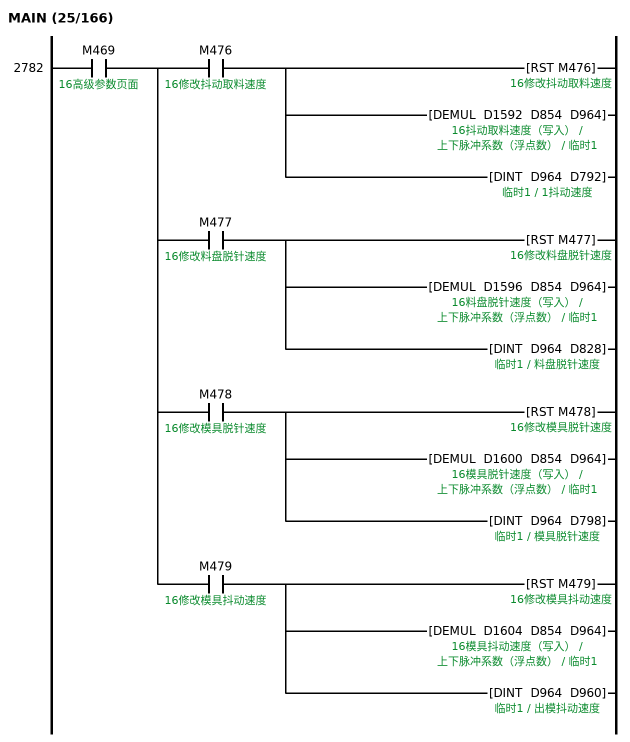
[picture p24: ladder of MAIN, rungs at steps 2782 to 2782]
2782  LD      M469  ; 16高级参数页面
      MPS
      AND     M476  ; 16修改抖动取料速度
      RST     M476  ; 16修改抖动取料速度
      DEMUL   D1592 D854 D964  ; 16抖动取料速度（写入）
      DINT    D964 D792
      MRD
      AND     M477  ; 16修改料盘脱针速度
      RST     M477  ; 16修改料盘脱针速度
      DEMUL   D1596 D854 D964  ; 16料盘脱针速度（写入）
      DINT    D964 D828
      MRD
      AND     M478  ; 16修改模具脱针速度
      RST     M478  ; 16修改模具脱针速度
      DEMUL   D1600 D854 D964  ; 16模具脱针速度（写入）
      DINT    D964 D798
      MPP
      AND     M479  ; 16修改模具抖动速度
      RST     M479  ; 16修改模具抖动速度
      DEMUL   D1604 D854 D964  ; 16模具抖动速度（写入）
      DINT    D964 D960
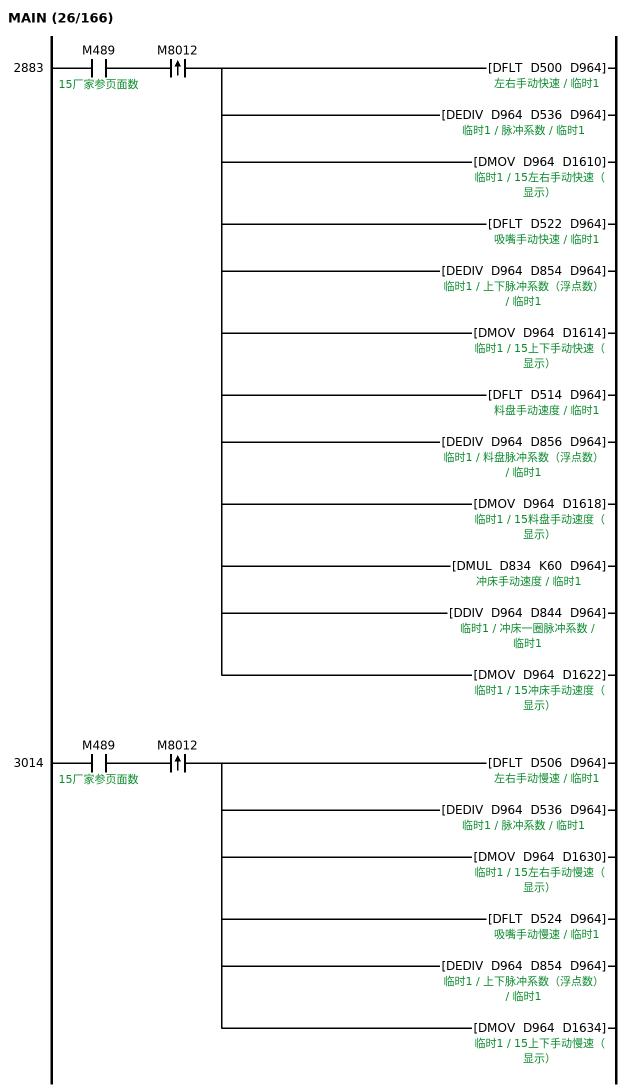
2883  LD      M489  ; 15厂家参页面数
      ANDP    M8012
      DFLT    D500 D964  ; 左右手动快速
      DEDIV   D964 D536 D964
      DMOV    D964 D1610  ; 15左右手动快速（显示）
      DFLT    D522 D964  ; 吸嘴手动快速
      DEDIV   D964 D854 D964
      DMOV    D964 D1614  ; 15上下手动快速（显示）
      DFLT    D514 D964  ; 料盘手动速度
      DEDIV   D964 D856 D964
      DMOV    D964 D1618  ; 15料盘手动速度（显示）
      DMUL    D834 K60 D964  ; 冲床手动速度
      DDIV    D964 D844 D964
      DMOV    D964 D1622  ; 15冲床手动速度（显示）
3014  LD      M489  ; 15厂家参页面数
      ANDP    M8012
      DFLT    D506 D964  ; 左右手动慢速
      DEDIV   D964 D536 D964
      DMOV    D964 D1630  ; 15左右手动慢速（显示）
      DFLT    D524 D964  ; 吸嘴手动慢速
      DEDIV   D964 D854 D964
      DMOV    D964 D1634  ; 15上下手动慢速（显示）
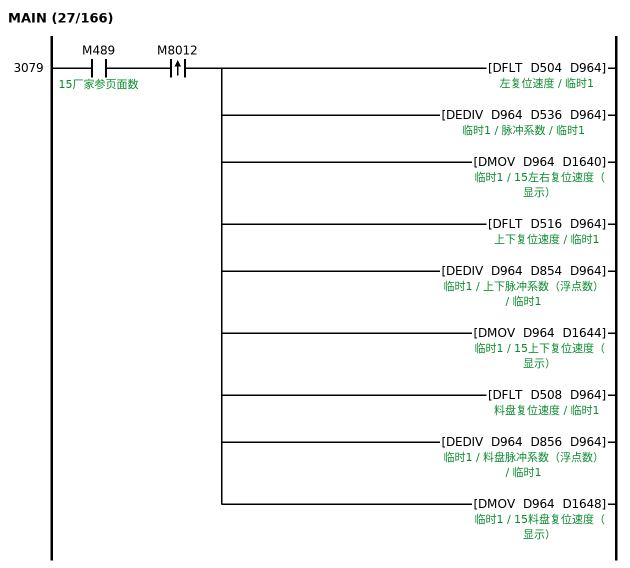
3079  LD      M489  ; 15厂家参页面数
      ANDP    M8012
      DFLT    D504 D964  ; 左复位速度
      DEDIV   D964 D536 D964
      DMOV    D964 D1640  ; 15左右复位速度（显示）
      DFLT    D516 D964  ; 上下复位速度
      DEDIV   D964 D854 D964
      DMOV    D964 D1644  ; 15上下复位速度（显示）
      DFLT    D508 D964  ; 料盘复位速度
      DEDIV   D964 D856 D964
      DMOV    D964 D1648  ; 15料盘复位速度（显示）
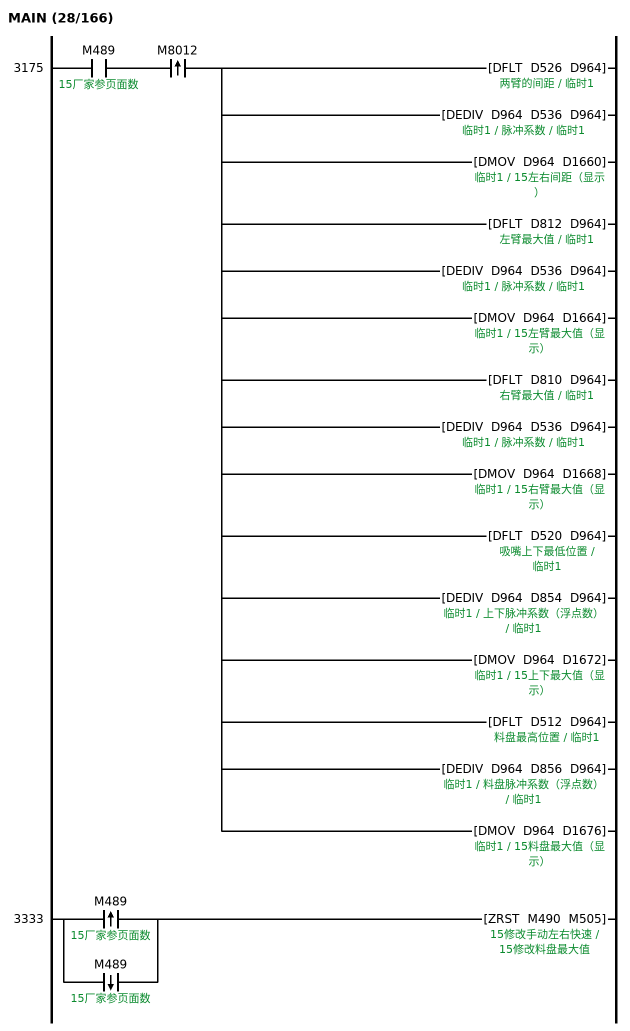
3175  LD      M489  ; 15厂家参页面数
      ANDP    M8012
      DFLT    D526 D964
      DEDIV   D964 D536 D964
      DMOV    D964 D1660  ; 15左右间距（显示）
      DFLT    D812 D964  ; 左臂最大值
      DEDIV   D964 D536 D964
      DMOV    D964 D1664  ; 15左臂最大值（显示）
      DFLT    D810 D964  ; 右臂最大值
      DEDIV   D964 D536 D964
      DMOV    D964 D1668  ; 15右臂最大值（显示）
      DFLT    D520 D964  ; 吸嘴上下最低位置
      DEDIV   D964 D854 D964
      DMOV    D964 D1672  ; 15上下最大值（显示）
      DFLT    D512 D964  ; 料盘最高位置
      DEDIV   D964 D856 D964
      DMOV    D964 D1676  ; 15料盘最大值（显示）
3333  LDP     M489  ; 15厂家参页面数
      ORF     M489  ; 15厂家参页面数
      ZRST    M490 M505  ; 15修改手动左右快速 / 15修改料盘最大值
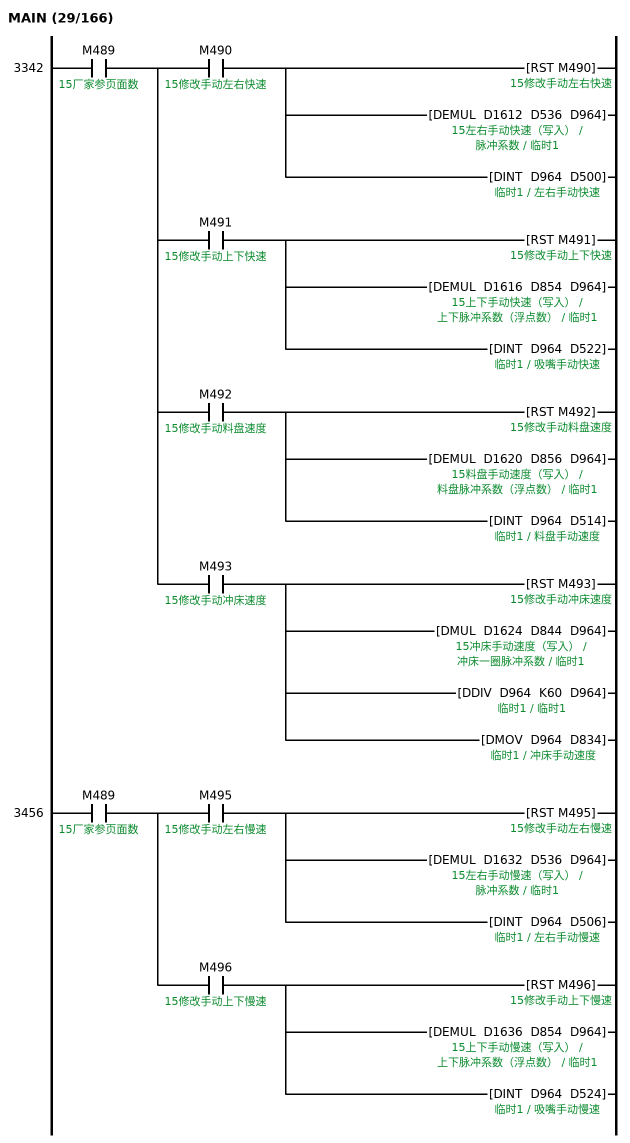
3342  LD      M489  ; 15厂家参页面数
      MPS
      AND     M490  ; 15修改手动左右快速
      RST     M490  ; 15修改手动左右快速
      DEMUL   D1612 D536 D964  ; 15左右手动快速（写入）
      DINT    D964 D500
      MRD
      AND     M491  ; 15修改手动上下快速
      RST     M491  ; 15修改手动上下快速
      DEMUL   D1616 D854 D964  ; 15上下手动快速（写入）
      DINT    D964 D522
      MRD
      AND     M492  ; 15修改手动料盘速度
      RST     M492  ; 15修改手动料盘速度
      DEMUL   D1620 D856 D964  ; 15料盘手动速度（写入）
      DINT    D964 D514
      MPP
      AND     M493  ; 15修改手动冲床速度
      RST     M493  ; 15修改手动冲床速度
      DMUL    D1624 D844 D964  ; 15冲床手动速度（写入）
      DDIV    D964 K60 D964
      DMOV    D964 D834
3456  LD      M489  ; 15厂家参页面数
      MPS
      AND     M495  ; 15修改手动左右慢速
      RST     M495  ; 15修改手动左右慢速
      DEMUL   D1632 D536 D964  ; 15左右手动慢速（写入）
      DINT    D964 D506
      MPP
      AND     M496  ; 15修改手动上下慢速
      RST     M496  ; 15修改手动上下慢速
      DEMUL   D1636 D854 D964  ; 15上下手动慢速（写入）
      DINT    D964 D524
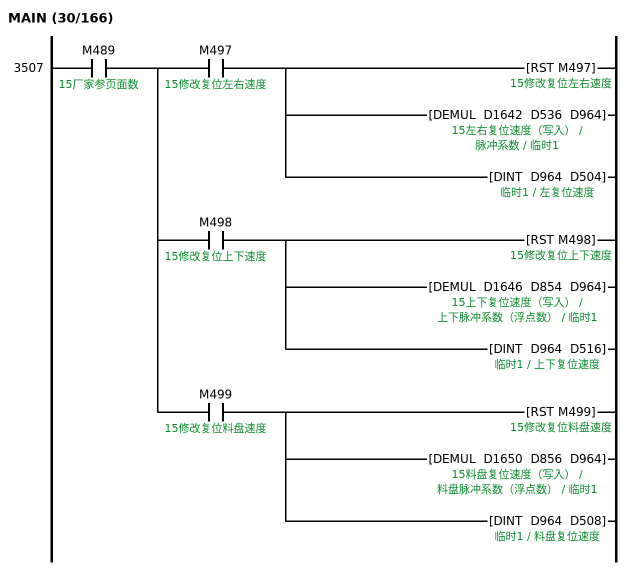
3507  LD      M489  ; 15厂家参页面数
      MPS
      AND     M497  ; 15修改复位左右速度
      RST     M497  ; 15修改复位左右速度
      DEMUL   D1642 D536 D964  ; 15左右复位速度（写入）
      DINT    D964 D504
      MRD
      AND     M498  ; 15修改复位上下速度
      RST     M498  ; 15修改复位上下速度
      DEMUL   D1646 D854 D964  ; 15上下复位速度（写入）
      DINT    D964 D516
      MPP
      AND     M499  ; 15修改复位料盘速度
      RST     M499  ; 15修改复位料盘速度
      DEMUL   D1650 D856 D964  ; 15料盘复位速度（写入）
      DINT    D964 D508
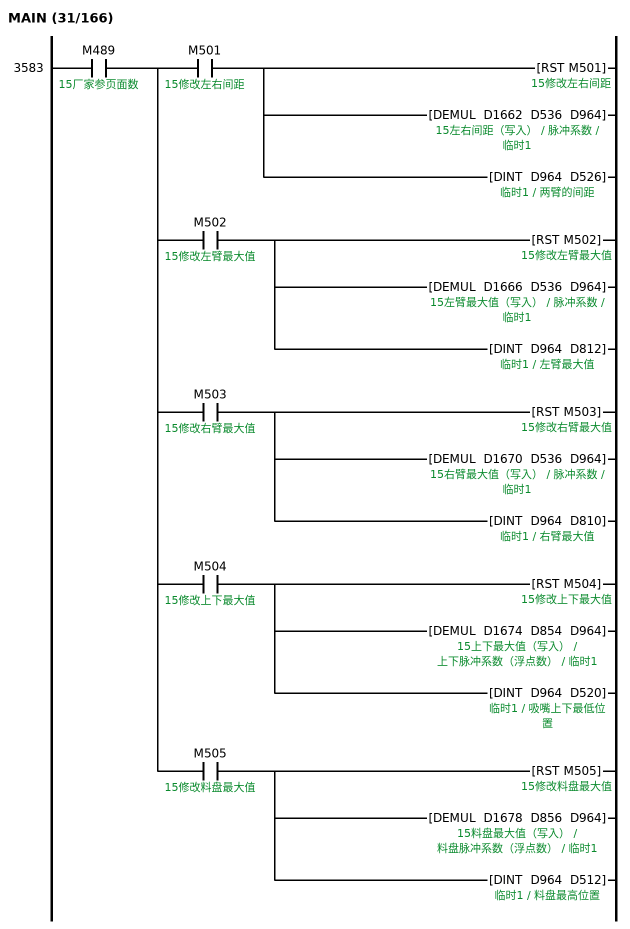
3583  LD      M489  ; 15厂家参页面数
      MPS
      AND     M501  ; 15修改左右间距
      RST     M501  ; 15修改左右间距
      DEMUL   D1662 D536 D964  ; 15左右间距（写入）
      DINT    D964 D526
      MRD
      AND     M502  ; 15修改左臂最大值
      RST     M502  ; 15修改左臂最大值
      DEMUL   D1666 D536 D964  ; 15左臂最大值（写入）
      DINT    D964 D812
      MRD
      AND     M503  ; 15修改右臂最大值
      RST     M503  ; 15修改右臂最大值
      DEMUL   D1670 D536 D964  ; 15右臂最大值（写入）
      DINT    D964 D810
      MRD
      AND     M504  ; 15修改上下最大值
      RST     M504  ; 15修改上下最大值
      DEMUL   D1674 D854 D964  ; 15上下最大值（写入）
      DINT    D964 D520
      MPP
      AND     M505  ; 15修改料盘最大值
      RST     M505  ; 15修改料盘最大值
      DEMUL   D1678 D856 D964  ; 15料盘最大值（写入）
      DINT    D964 D512
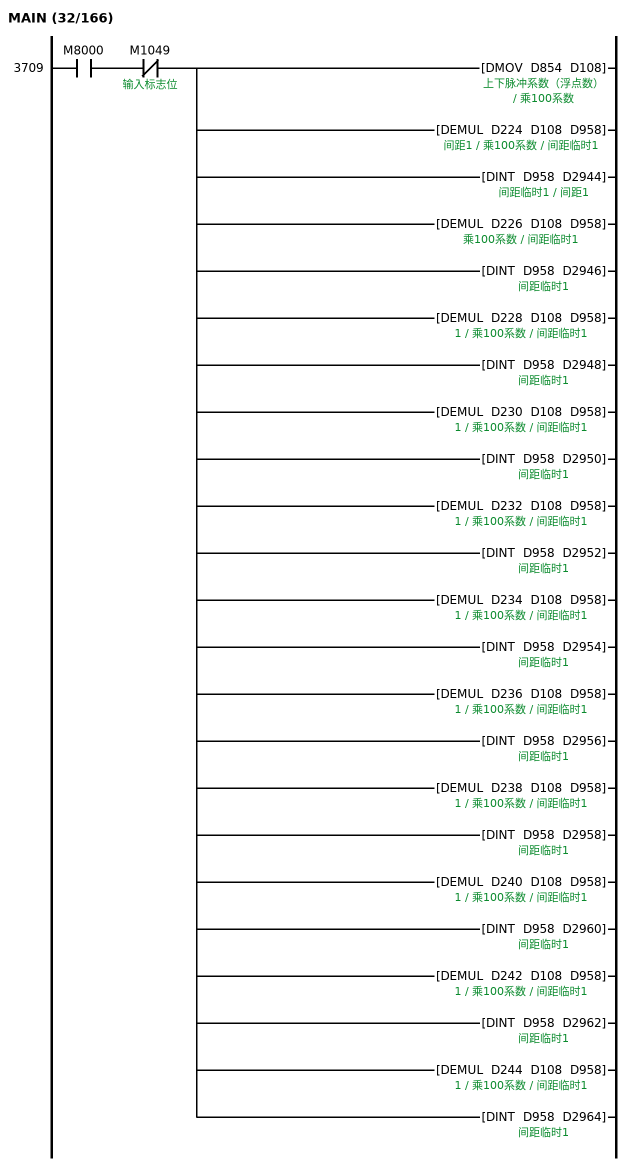
3709  LD      M8000
      ANI     M1049  ; 输入标志位
      DMOV    D854 D108  ; 乘100系数
      DEMUL   D224 D108 D958  ; 间距1 / 间距临时1
      DINT    D958 D2944  ; 间距1
      DEMUL   D226 D108 D958
      DINT    D958 D2946
      DEMUL   D228 D108 D958  ; 1
      DINT    D958 D2948
      DEMUL   D230 D108 D958  ; 1
      DINT    D958 D2950
      DEMUL   D232 D108 D958  ; 1
      DINT    D958 D2952
      DEMUL   D234 D108 D958  ; 1
      DINT    D958 D2954
      DEMUL   D236 D108 D958  ; 1
      DINT    D958 D2956
      DEMUL   D238 D108 D958  ; 1
      DINT    D958 D2958
      DEMUL   D240 D108 D958  ; 1
      DINT    D958 D2960
      DEMUL   D242 D108 D958  ; 1
      DINT    D958 D2962
      DEMUL   D244 D108 D958  ; 1
      DINT    D958 D2964
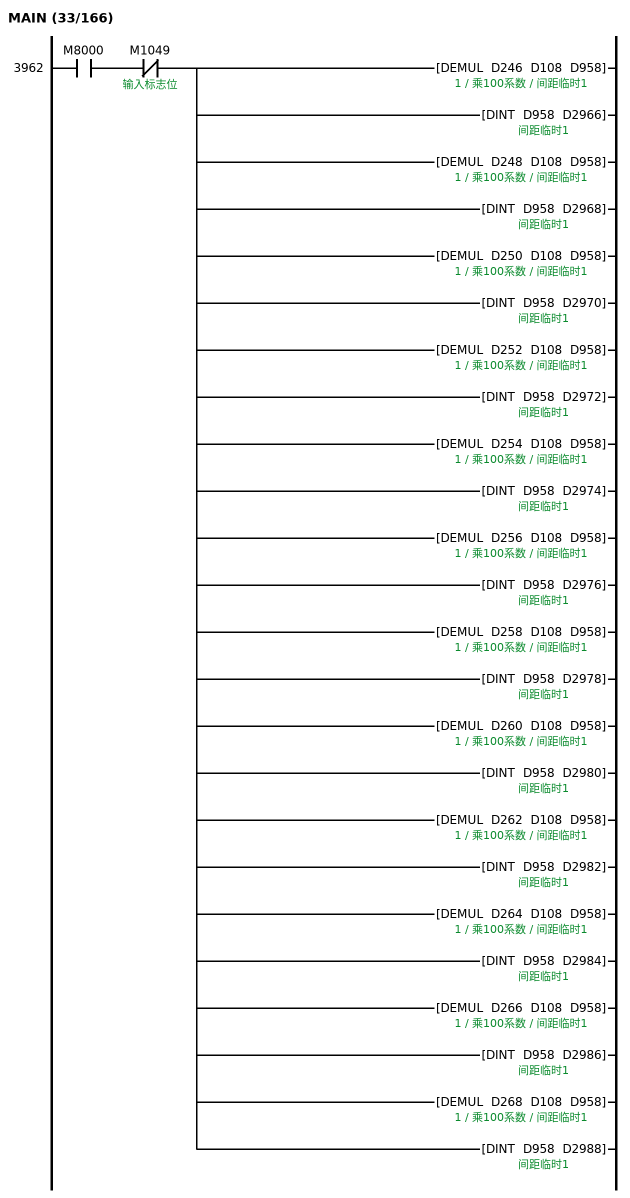
3962  LD      M8000
      ANI     M1049  ; 输入标志位
      DEMUL   D246 D108 D958  ; 1
      DINT    D958 D2966
      DEMUL   D248 D108 D958  ; 1
      DINT    D958 D2968
      DEMUL   D250 D108 D958  ; 1
      DINT    D958 D2970
      DEMUL   D252 D108 D958  ; 1
      DINT    D958 D2972
      DEMUL   D254 D108 D958  ; 1
      DINT    D958 D2974
      DEMUL   D256 D108 D958  ; 1
      DINT    D958 D2976
      DEMUL   D258 D108 D958  ; 1
      DINT    D958 D2978
      DEMUL   D260 D108 D958  ; 1
      DINT    D958 D2980
      DEMUL   D262 D108 D958  ; 1
      DINT    D958 D2982
      DEMUL   D264 D108 D958  ; 1
      DINT    D958 D2984
      DEMUL   D266 D108 D958  ; 1
      DINT    D958 D2986
      DEMUL   D268 D108 D958  ; 1
      DINT    D958 D2988
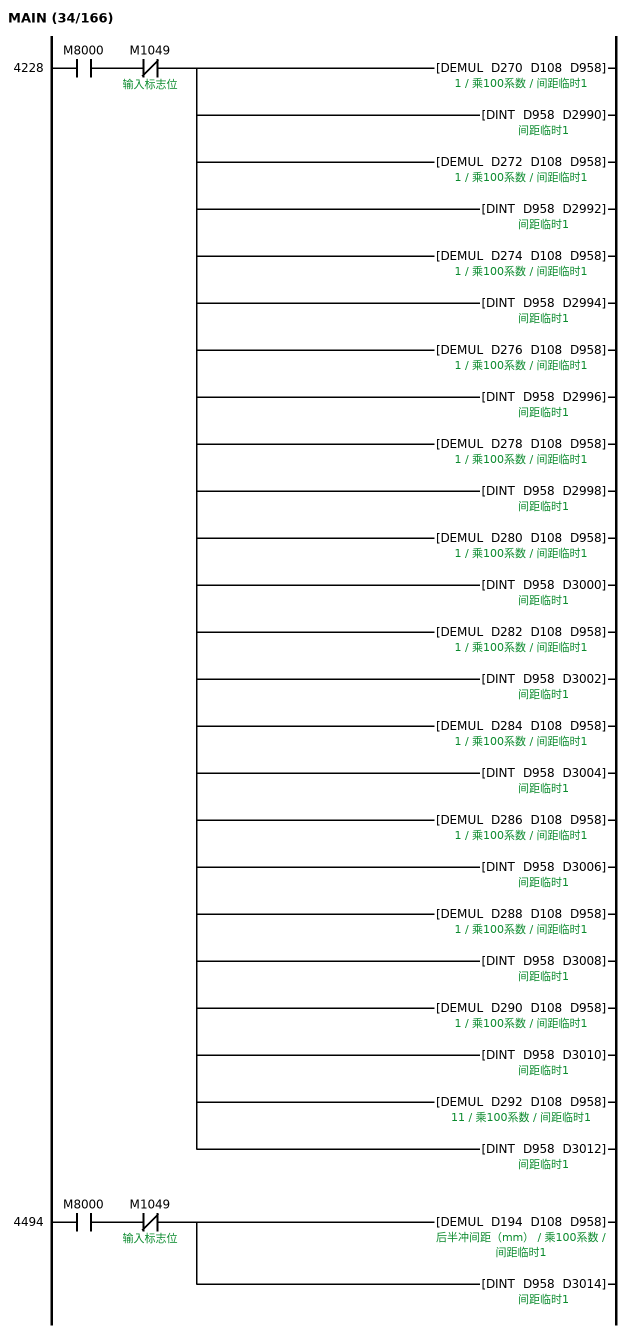
4228  LD      M8000
      ANI     M1049  ; 输入标志位
      DEMUL   D270 D108 D958  ; 1
      DINT    D958 D2990
      DEMUL   D272 D108 D958  ; 1
      DINT    D958 D2992
      DEMUL   D274 D108 D958  ; 1
      DINT    D958 D2994
      DEMUL   D276 D108 D958  ; 1
      DINT    D958 D2996
      DEMUL   D278 D108 D958  ; 1
      DINT    D958 D2998
      DEMUL   D280 D108 D958  ; 1
      DINT    D958 D3000
      DEMUL   D282 D108 D958  ; 1
      DINT    D958 D3002
      DEMUL   D284 D108 D958  ; 1
      DINT    D958 D3004
      DEMUL   D286 D108 D958  ; 1
      DINT    D958 D3006
      DEMUL   D288 D108 D958  ; 1
      DINT    D958 D3008
      DEMUL   D290 D108 D958  ; 1
      DINT    D958 D3010
      DEMUL   D292 D108 D958  ; 11
      DINT    D958 D3012
4494  LD      M8000
      ANI     M1049  ; 输入标志位
      DEMUL   D194 D108 D958
      DINT    D958 D3014
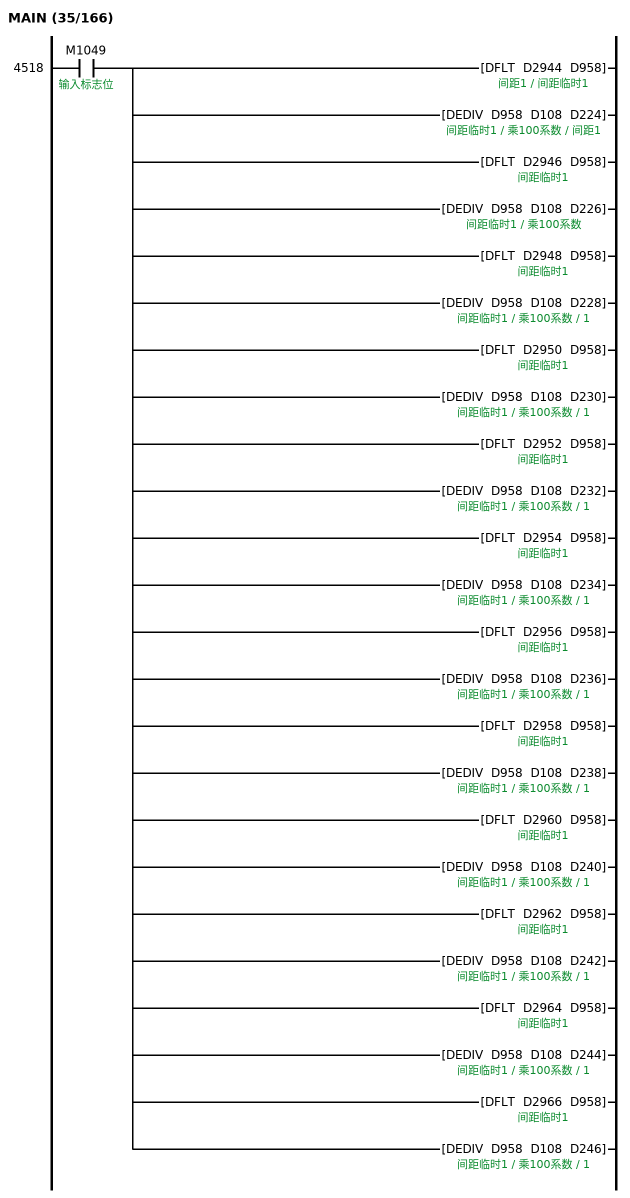
4518  LD      M1049  ; 输入标志位
      DFLT    D2944 D958
      DEDIV   D958 D108 D224
      DFLT    D2946 D958
      DEDIV   D958 D108 D226
      DFLT    D2948 D958
      DEDIV   D958 D108 D228
      DFLT    D2950 D958
      DEDIV   D958 D108 D230
      DFLT    D2952 D958
      DEDIV   D958 D108 D232
      DFLT    D2954 D958
      DEDIV   D958 D108 D234
      DFLT    D2956 D958
      DEDIV   D958 D108 D236
      DFLT    D2958 D958
      DEDIV   D958 D108 D238
      DFLT    D2960 D958
      DEDIV   D958 D108 D240
      DFLT    D2962 D958
      DEDIV   D958 D108 D242
      DFLT    D2964 D958
      DEDIV   D958 D108 D244
      DFLT    D2966 D958
      DEDIV   D958 D108 D246
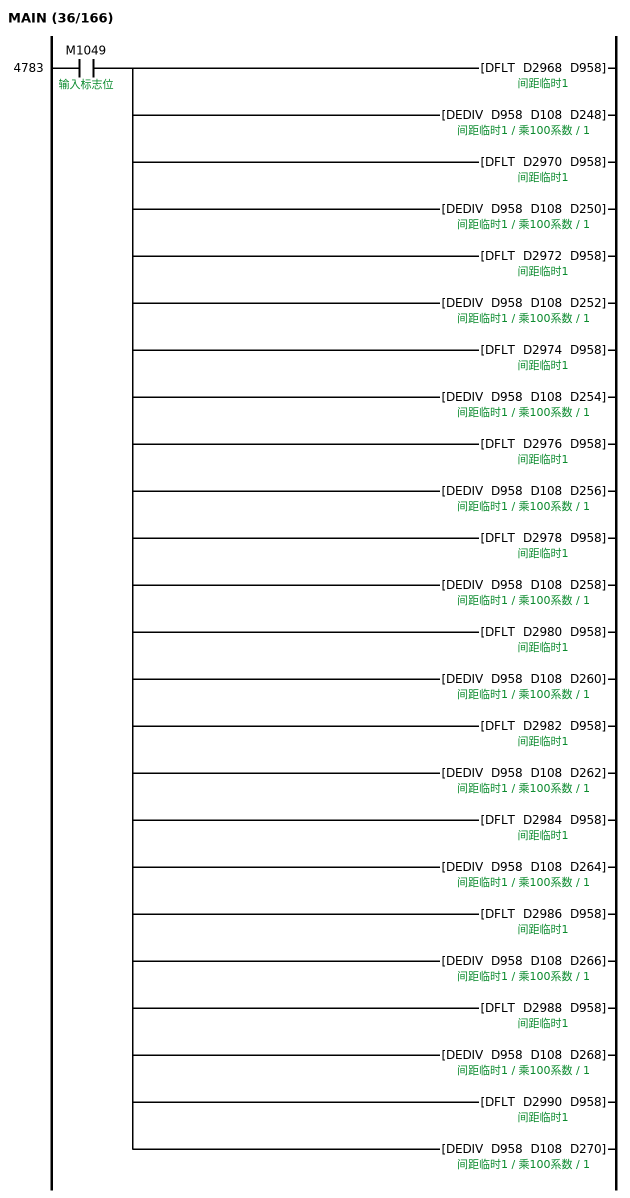
4783  LD      M1049  ; 输入标志位
      DFLT    D2968 D958
      DEDIV   D958 D108 D248
      DFLT    D2970 D958
      DEDIV   D958 D108 D250
      DFLT    D2972 D958
      DEDIV   D958 D108 D252
      DFLT    D2974 D958
      DEDIV   D958 D108 D254
      DFLT    D2976 D958
      DEDIV   D958 D108 D256
      DFLT    D2978 D958
      DEDIV   D958 D108 D258
      DFLT    D2980 D958
      DEDIV   D958 D108 D260
      DFLT    D2982 D958
      DEDIV   D958 D108 D262
      DFLT    D2984 D958
      DEDIV   D958 D108 D264
      DFLT    D2986 D958
      DEDIV   D958 D108 D266
      DFLT    D2988 D958
      DEDIV   D958 D108 D268
      DFLT    D2990 D958
      DEDIV   D958 D108 D270
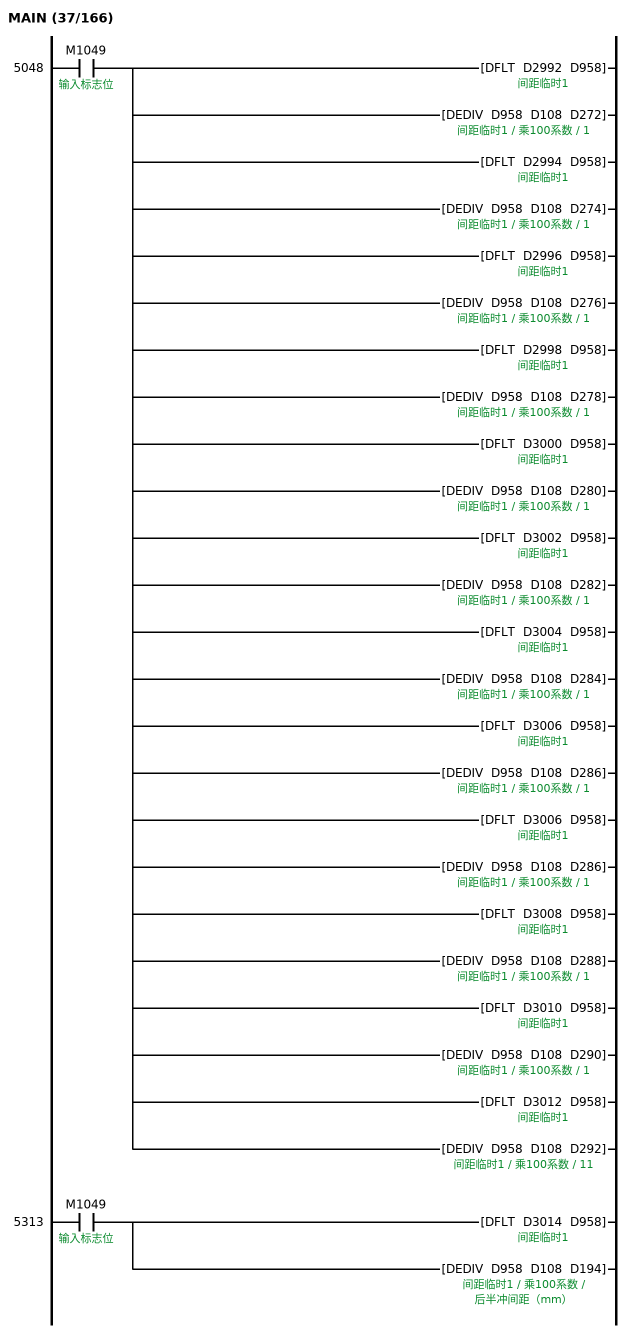
5048  LD      M1049  ; 输入标志位
      DFLT    D2992 D958
      DEDIV   D958 D108 D272
      DFLT    D2994 D958
      DEDIV   D958 D108 D274
      DFLT    D2996 D958
      DEDIV   D958 D108 D276
      DFLT    D2998 D958
      DEDIV   D958 D108 D278
      DFLT    D3000 D958
      DEDIV   D958 D108 D280
      DFLT    D3002 D958
      DEDIV   D958 D108 D282
      DFLT    D3004 D958
      DEDIV   D958 D108 D284
      DFLT    D3006 D958
      DEDIV   D958 D108 D286
      DFLT    D3006 D958
      DEDIV   D958 D108 D286
      DFLT    D3008 D958
      DEDIV   D958 D108 D288
      DFLT    D3010 D958
      DEDIV   D958 D108 D290
      DFLT    D3012 D958
      DEDIV   D958 D108 D292
5313  LD      M1049  ; 输入标志位
      DFLT    D3014 D958
      DEDIV   D958 D108 D194
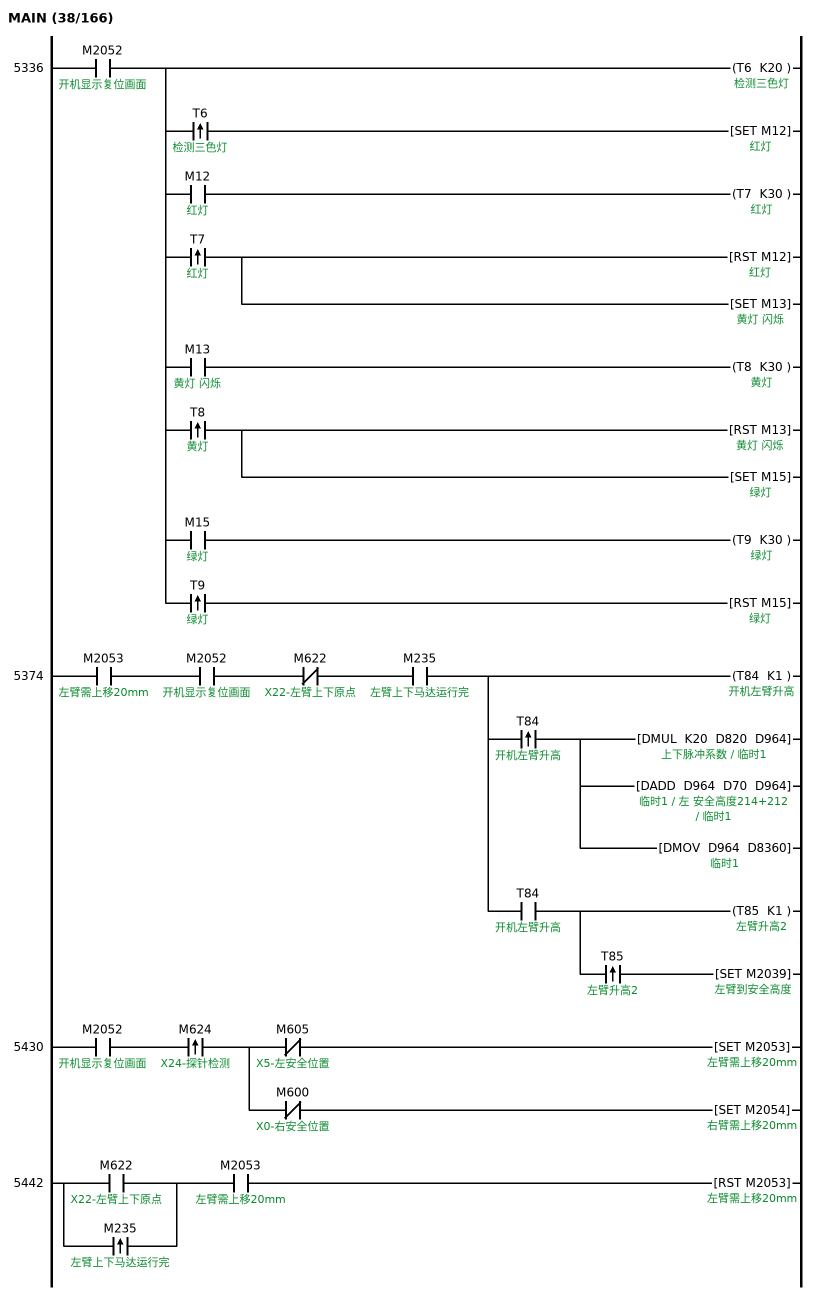
5336  LD      M2052  ; 开机显示复位画面
      OUT     T6 K20  ; 检测三色灯
      MPS
      ANDP    T6  ; 检测三色灯
      SET     M12  ; 红灯
      MRD
      AND     M12  ; 红灯
      OUT     T7 K30  ; 红灯
      MRD
      ANDP    T7  ; 红灯
      RST     M12  ; 红灯
      SET     M13  ; 黄灯 闪烁
      MRD
      AND     M13  ; 黄灯 闪烁
      OUT     T8 K30  ; 黄灯
      MRD
      ANDP    T8  ; 黄灯
      RST     M13  ; 黄灯 闪烁
      SET     M15  ; 绿灯
      MRD
      AND     M15  ; 绿灯
      OUT     T9 K30  ; 绿灯
      MPP
      ANDP    T9  ; 绿灯
      RST     M15  ; 绿灯
5374  LD      M2053  ; 左臂需上移20mm
      AND     M2052  ; 开机显示复位画面
      ANI     M622  ; X22-左臂上下原点
      AND     M235  ; 左臂上下马达运行完
      OUT     T84 K1  ; 开机左臂升高
      MPS
      ANDP    T84  ; 开机左臂升高
      DMUL    K20 D820 D964
      DADD    D964 D70 D964
      DMOV    D964 D8360
      MPP
      AND     T84  ; 开机左臂升高
      OUT     T85 K1  ; 左臂升高2
      ANDP    T85  ; 左臂升高2
      SET     M2039  ; 左臂到安全高度
5430  LD      M2052  ; 开机显示复位画面
      ANDP    M624  ; X24-探针检测
      MPS
      ANI     M605  ; X5-左安全位置
      SET     M2053  ; 左臂需上移20mm
      MPP
      ANI     M600  ; X0-右安全位置
      SET     M2054  ; 右臂需上移20mm
5442  LD      M622  ; X22-左臂上下原点
      ORP     M235  ; 左臂上下马达运行完
      AND     M2053  ; 左臂需上移20mm
      RST     M2053  ; 左臂需上移20mm
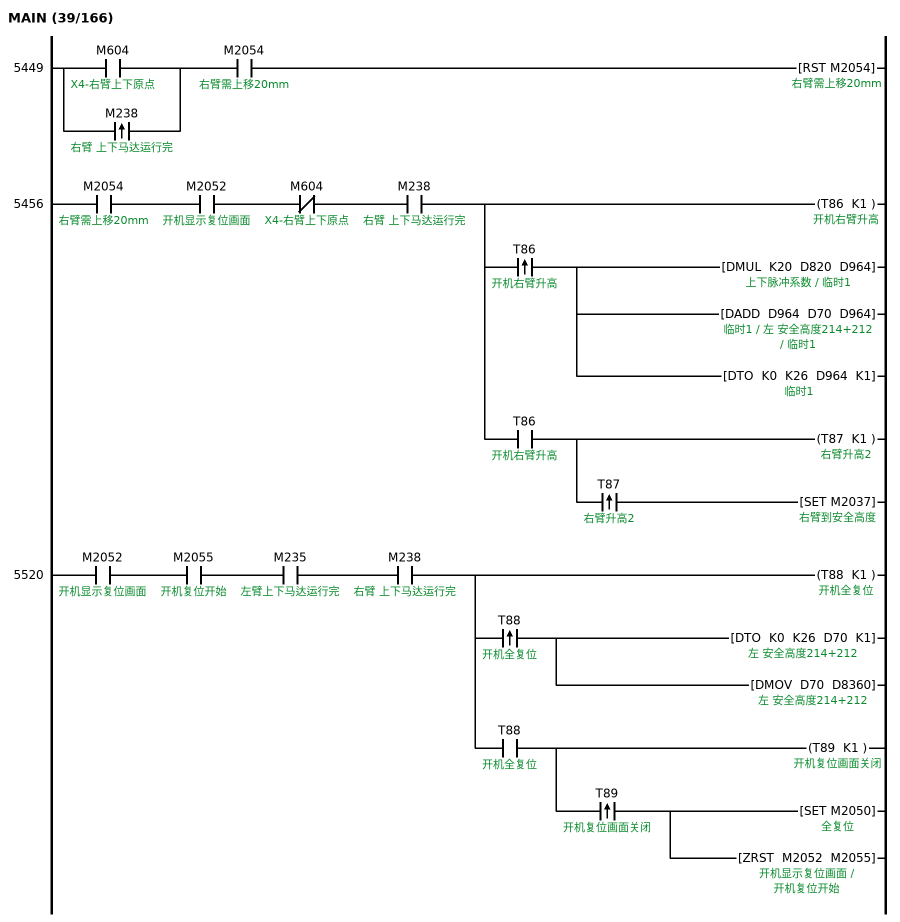
5449  LD      M604  ; X4-右臂上下原点
      ORP     M238  ; 右臂 上下马达运行完
      AND     M2054  ; 右臂需上移20mm
      RST     M2054  ; 右臂需上移20mm
5456  LD      M2054  ; 右臂需上移20mm
      AND     M2052  ; 开机显示复位画面
      ANI     M604  ; X4-右臂上下原点
      AND     M238  ; 右臂 上下马达运行完
      OUT     T86 K1  ; 开机右臂升高
      MPS
      ANDP    T86  ; 开机右臂升高
      DMUL    K20 D820 D964
      DADD    D964 D70 D964
      DTO     K0 K26 D964 K1
      MPP
      AND     T86  ; 开机右臂升高
      OUT     T87 K1  ; 右臂升高2
      ANDP    T87  ; 右臂升高2
      SET     M2037  ; 右臂到安全高度
5520  LD      M2052  ; 开机显示复位画面
      AND     M2055  ; 开机复位开始
      AND     M235  ; 左臂上下马达运行完
      AND     M238  ; 右臂 上下马达运行完
      OUT     T88 K1  ; 开机全复位
      MPS
      ANDP    T88  ; 开机全复位
      DTO     K0 K26 D70 K1
      DMOV    D70 D8360
      MPP
      AND     T88  ; 开机全复位
      OUT     T89 K1  ; 开机复位画面关闭
      ANDP    T89  ; 开机复位画面关闭
      SET     M2050  ; 全复位
      ZRST    M2052 M2055
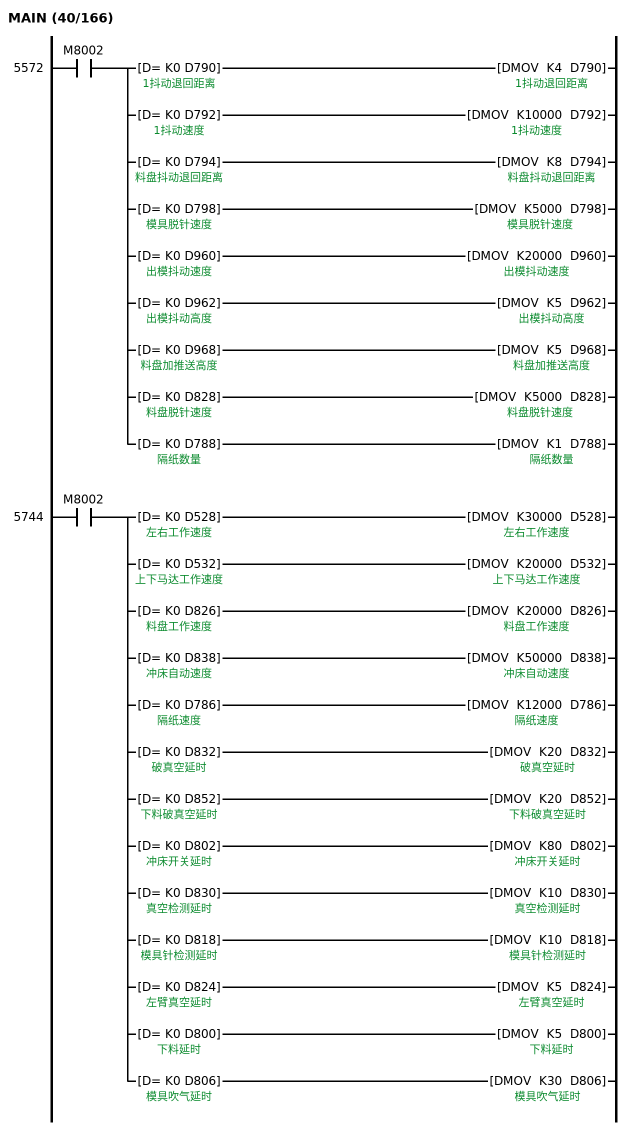
5572  LD      M8002
      MPS
      ANDD=   K0 D790  ; 1抖动退回距离
      DMOV    K4 D790
      MRD
      ANDD=   K0 D792  ; 1抖动速度
      DMOV    K10000 D792
      MRD
      ANDD=   K0 D794  ; 料盘抖动退回距离
      DMOV    K8 D794
      MRD
      ANDD=   K0 D798  ; 模具脱针速度
      DMOV    K5000 D798
      MRD
      ANDD=   K0 D960  ; 出模抖动速度
      DMOV    K20000 D960
      MRD
      ANDD=   K0 D962  ; 出模抖动高度
      DMOV    K5 D962
      MRD
      ANDD=   K0 D968  ; 料盘加推送高度
      DMOV    K5 D968
      MRD
      ANDD=   K0 D828  ; 料盘脱针速度
      DMOV    K5000 D828
      MPP
      ANDD=   K0 D788  ; 隔纸数量
      DMOV    K1 D788
5744  LD      M8002
      MPS
      ANDD=   K0 D528  ; 左右工作速度
      DMOV    K30000 D528
      MRD
      ANDD=   K0 D532  ; 上下马达工作速度
      DMOV    K20000 D532
      MRD
      ANDD=   K0 D826  ; 料盘工作速度
      DMOV    K20000 D826
      MRD
      ANDD=   K0 D838  ; 冲床自动速度
      DMOV    K50000 D838
      MRD
      ANDD=   K0 D786  ; 隔纸速度
      DMOV    K12000 D786
      MRD
      ANDD=   K0 D832  ; 破真空延时
      DMOV    K20 D832
      MRD
      ANDD=   K0 D852  ; 下料破真空延时
      DMOV    K20 D852
      MRD
      ANDD=   K0 D802  ; 冲床开关延时
      DMOV    K80 D802
      MRD
      ANDD=   K0 D830  ; 真空检测延时
      DMOV    K10 D830
      MRD
      ANDD=   K0 D818  ; 模具针检测延时
      DMOV    K10 D818
      MRD
      ANDD=   K0 D824  ; 左臂真空延时
      DMOV    K5 D824
      MRD
      ANDD=   K0 D800  ; 下料延时
      DMOV    K5 D800
      MPP
      ANDD=   K0 D806  ; 模具吹气延时
      DMOV    K30 D806
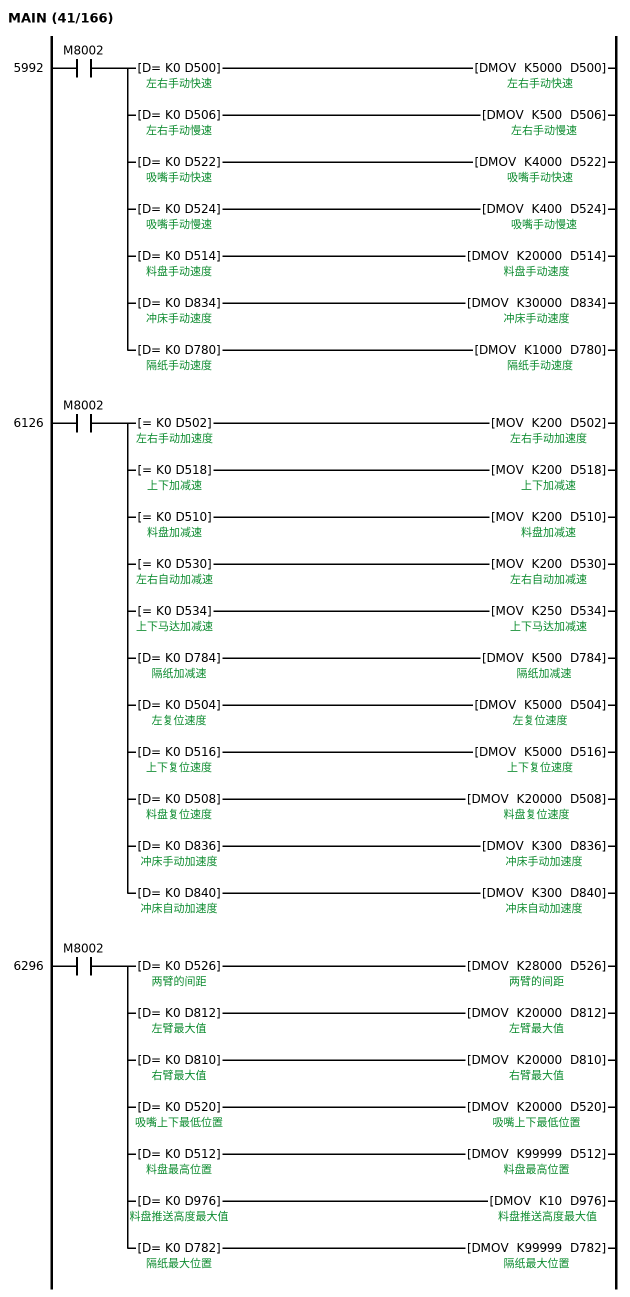
5992  LD      M8002
      MPS
      ANDD=   K0 D500  ; 左右手动快速
      DMOV    K5000 D500
      MRD
      ANDD=   K0 D506  ; 左右手动慢速
      DMOV    K500 D506
      MRD
      ANDD=   K0 D522  ; 吸嘴手动快速
      DMOV    K4000 D522
      MRD
      ANDD=   K0 D524  ; 吸嘴手动慢速
      DMOV    K400 D524
      MRD
      ANDD=   K0 D514  ; 料盘手动速度
      DMOV    K20000 D514
      MRD
      ANDD=   K0 D834  ; 冲床手动速度
      DMOV    K30000 D834
      MPP
      ANDD=   K0 D780  ; 隔纸手动速度
      DMOV    K1000 D780
6126  LD      M8002
      MPS
      AND=    K0 D502  ; 左右手动加速度
      MOV     K200 D502
      MRD
      AND=    K0 D518  ; 上下加减速
      MOV     K200 D518
      MRD
      AND=    K0 D510  ; 料盘加减速
      MOV     K200 D510
      MRD
      AND=    K0 D530  ; 左右自动加减速
      MOV     K200 D530
      MRD
      AND=    K0 D534  ; 上下马达加减速
      MOV     K250 D534
      MRD
      ANDD=   K0 D784  ; 隔纸加减速
      DMOV    K500 D784
      MRD
      ANDD=   K0 D504  ; 左复位速度
      DMOV    K5000 D504
      MRD
      ANDD=   K0 D516  ; 上下复位速度
      DMOV    K5000 D516
      MRD
      ANDD=   K0 D508  ; 料盘复位速度
      DMOV    K20000 D508
      MRD
      ANDD=   K0 D836  ; 冲床手动加速度
      DMOV    K300 D836
      MPP
      ANDD=   K0 D840  ; 冲床自动加速度
      DMOV    K300 D840
6296  LD      M8002
      MPS
      ANDD=   K0 D526  ; 两臂的间距
      DMOV    K28000 D526
      MRD
      ANDD=   K0 D812  ; 左臂最大值
      DMOV    K20000 D812
      MRD
      ANDD=   K0 D810  ; 右臂最大值
      DMOV    K20000 D810
      MRD
      ANDD=   K0 D520  ; 吸嘴上下最低位置
      DMOV    K20000 D520
      MRD
      ANDD=   K0 D512  ; 料盘最高位置
      DMOV    K99999 D512
      MRD
      ANDD=   K0 D976  ; 料盘推送高度最大值
      DMOV    K10 D976
      MPP
      ANDD=   K0 D782  ; 隔纸最大位置
      DMOV    K99999 D782
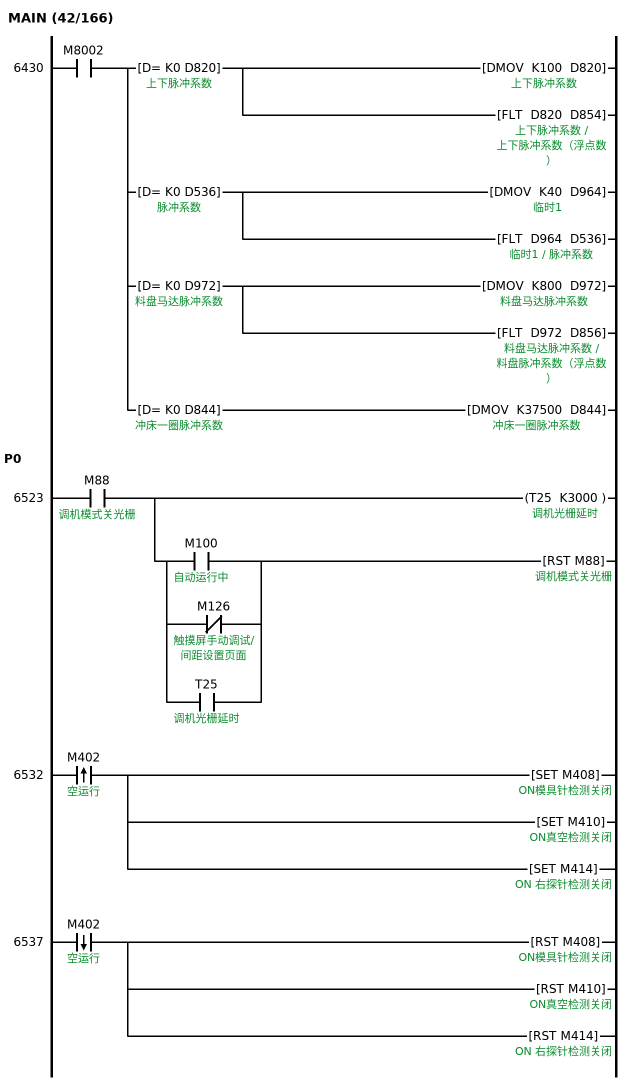
6430  LD      M8002
      MPS
      ANDD=   K0 D820  ; 上下脉冲系数
      DMOV    K100 D820
      FLT     D820 D854
      MRD
      ANDD=   K0 D536  ; 脉冲系数
      DMOV    K40 D964
      FLT     D964 D536
      MRD
      ANDD=   K0 D972  ; 料盘马达脉冲系数
      DMOV    K800 D972
      FLT     D972 D856
      MPP
      ANDD=   K0 D844  ; 冲床一圈脉冲系数
      DMOV    K37500 D844
      P0
6523  LD      M88  ; 调机模式关光栅
      OUT     T25 K3000  ; 调机光栅延时
      LD      M100  ; 自动运行中
      ORI     M126  ; 触摸屏手动调试/间距设置页面
      OR      T25  ; 调机光栅延时
      ANB
      RST     M88  ; 调机模式关光栅
6532  LDP     M402  ; 空运行
      SET     M408  ; ON模具针检测关闭
      SET     M410  ; ON真空检测关闭
      SET     M414  ; ON 右探针检测关闭
6537  LDF     M402  ; 空运行
      RST     M408  ; ON模具针检测关闭
      RST     M410  ; ON真空检测关闭
      RST     M414  ; ON 右探针检测关闭
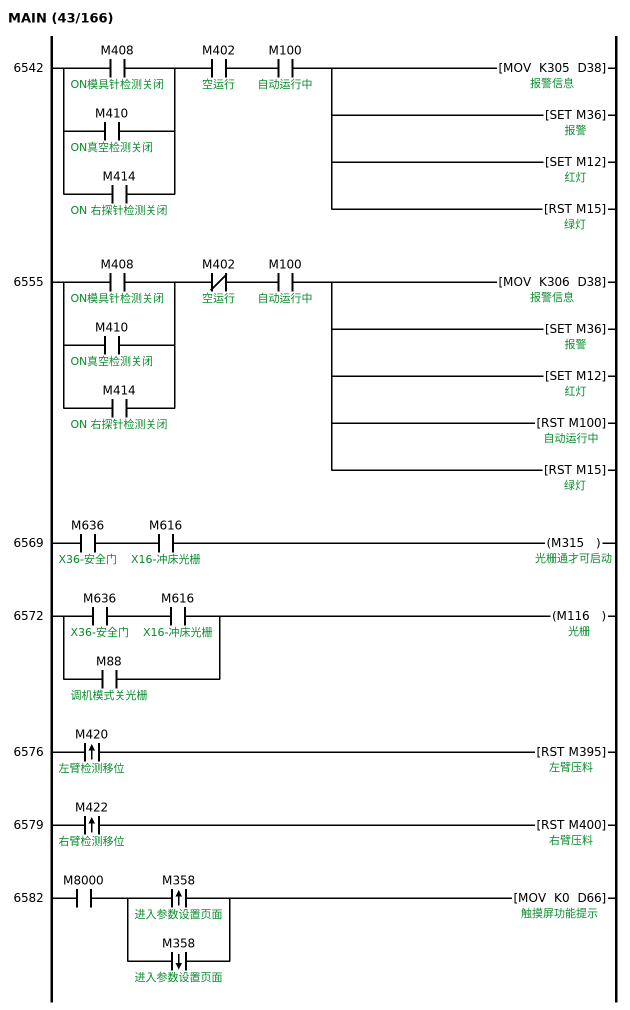
6542  LD      M408  ; ON模具针检测关闭
      OR      M410  ; ON真空检测关闭
      OR      M414  ; ON 右探针检测关闭
      AND     M402  ; 空运行
      AND     M100  ; 自动运行中
      MOV     K305 D38
      SET     M36  ; 报警
      SET     M12  ; 红灯
      RST     M15  ; 绿灯
6555  LD      M408  ; ON模具针检测关闭
      OR      M410  ; ON真空检测关闭
      OR      M414  ; ON 右探针检测关闭
      ANI     M402  ; 空运行
      AND     M100  ; 自动运行中
      MOV     K306 D38
      SET     M36  ; 报警
      SET     M12  ; 红灯
      RST     M100  ; 自动运行中
      RST     M15  ; 绿灯
6569  LD      M636  ; X36-安全门
      AND     M616  ; X16-冲床光栅
      OUT     M315  ; 光栅通才可启动
6572  LD      M636  ; X36-安全门
      AND     M616  ; X16-冲床光栅
      OR      M88  ; 调机模式关光栅
      OUT     M116  ; 光栅
6576  LDP     M420  ; 左臂检测移位
      RST     M395  ; 左臂压料
6579  LDP     M422  ; 右臂检测移位
      RST     M400  ; 右臂压料
6582  LD      M8000
      LDP     M358  ; 进入参数设置页面
      ORF     M358  ; 进入参数设置页面
      ANB
      MOV     K0 D66  ; 触摸屏功能提示
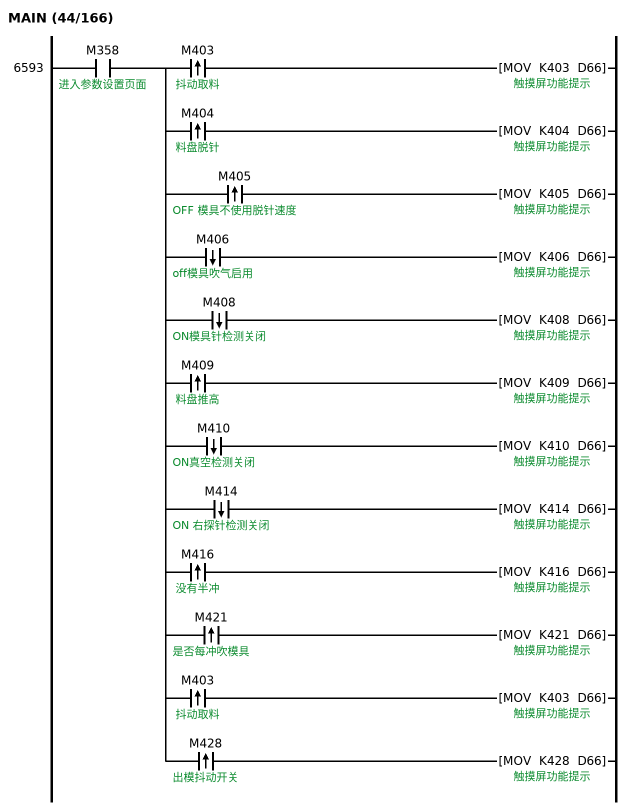
6593  LD      M358  ; 进入参数设置页面
      MPS
      ANDP    M403  ; 抖动取料
      MOV     K403 D66
      MRD
      ANDP    M404  ; 料盘脱针
      MOV     K404 D66
      MRD
      ANDP    M405  ; OFF 模具不使用脱针速度
      MOV     K405 D66
      MRD
      ANDF    M406  ; off模具吹气启用
      MOV     K406 D66
      MRD
      ANDF    M408  ; ON模具针检测关闭
      MOV     K408 D66
      MRD
      ANDP    M409  ; 料盘推高
      MOV     K409 D66
      MRD
      ANDF    M410  ; ON真空检测关闭
      MOV     K410 D66
      MRD
      ANDF    M414  ; ON 右探针检测关闭
      MOV     K414 D66
      MRD
      ANDP    M416  ; 没有半冲
      MOV     K416 D66
      MRD
      ANDP    M421  ; 是否每冲吹模具
      MOV     K421 D66
      MRD
      ANDP    M403  ; 抖动取料
      MOV     K403 D66
      MPP
      ANDP    M428  ; 出模抖动开关
      MOV     K428 D66
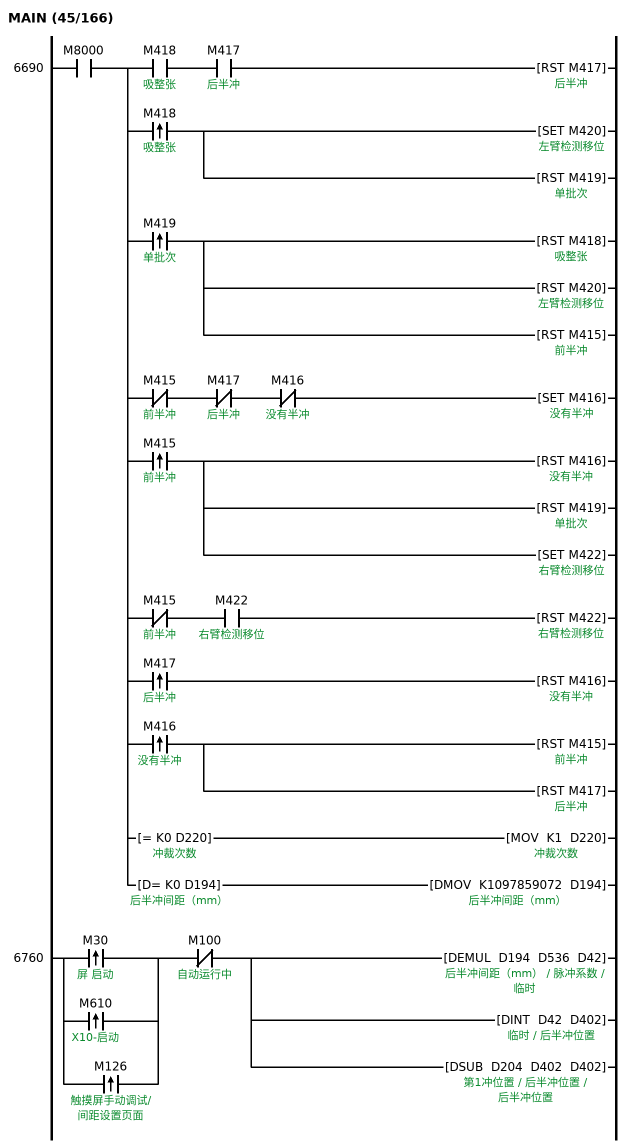
6690  LD      M8000
      MPS
      AND     M418  ; 吸整张
      AND     M417  ; 后半冲
      RST     M417  ; 后半冲
      MRD
      ANDP    M418  ; 吸整张
      SET     M420  ; 左臂检测移位
      RST     M419  ; 单批次
      MRD
      ANDP    M419  ; 单批次
      RST     M418  ; 吸整张
      RST     M420  ; 左臂检测移位
      RST     M415  ; 前半冲
      MRD
      ANI     M415  ; 前半冲
      ANI     M417  ; 后半冲
      ANI     M416  ; 没有半冲
      SET     M416  ; 没有半冲
      MRD
      ANDP    M415  ; 前半冲
      RST     M416  ; 没有半冲
      RST     M419  ; 单批次
      SET     M422  ; 右臂检测移位
      MRD
      ANI     M415  ; 前半冲
      AND     M422  ; 右臂检测移位
      RST     M422  ; 右臂检测移位
      MRD
      ANDP    M417  ; 后半冲
      RST     M416  ; 没有半冲
      MRD
      ANDP    M416  ; 没有半冲
      RST     M415  ; 前半冲
      RST     M417  ; 后半冲
      MRD
      AND=    K0 D220  ; 冲裁次数
      MOV     K1 D220
      MPP
      ANDD=   K0 D194  ; 后半冲间距（mm）
      DMOV    K1097859072 D194
6760  LDP     M30  ; 屏 启动
      ORP     M610  ; X10-启动
      ORP     M126  ; 触摸屏手动调试/间距设置页面
      ANI     M100  ; 自动运行中
      DEMUL   D194 D536 D42  ; 临时
      DINT    D42 D402  ; 后半冲位置
      DSUB    D204 D402 D402
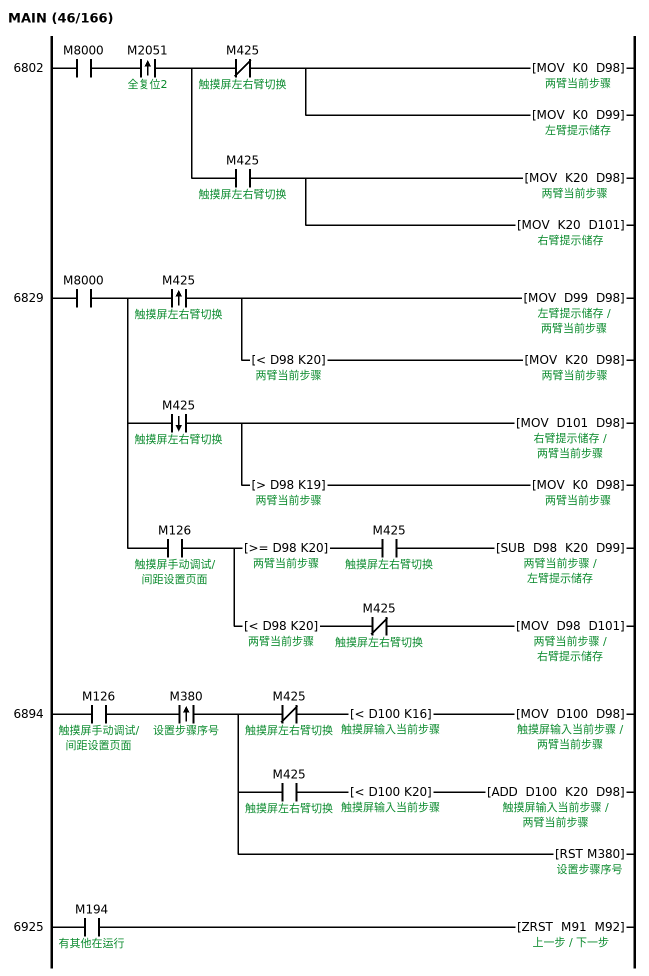
6802  LD      M8000
      ANDP    M2051  ; 全复位2
      MPS
      ANI     M425  ; 触摸屏左右臂切换
      MOV     K0 D98  ; 两臂当前步骤
      MOV     K0 D99  ; 左臂提示储存
      MPP
      AND     M425  ; 触摸屏左右臂切换
      MOV     K20 D98
      MOV     K20 D101  ; 右臂提示储存
6829  LD      M8000
      MPS
      ANDP    M425  ; 触摸屏左右臂切换
      MOV     D99 D98
      AND<    D98 K20  ; 两臂当前步骤
      MOV     K20 D98
      MRD
      ANDF    M425  ; 触摸屏左右臂切换
      MOV     D101 D98
      AND>    D98 K19  ; 两臂当前步骤
      MOV     K0 D98
      MPP
      AND     M126  ; 触摸屏手动调试/间距设置页面
      MPS
      AND>=   D98 K20  ; 两臂当前步骤
      AND     M425  ; 触摸屏左右臂切换
      SUB     D98 K20 D99
      MPP
      AND<    D98 K20  ; 两臂当前步骤
      ANI     M425  ; 触摸屏左右臂切换
      MOV     D98 D101
6894  LD      M126  ; 触摸屏手动调试/间距设置页面
      ANDP    M380  ; 设置步骤序号
      MPS
      ANI     M425  ; 触摸屏左右臂切换
      AND<    D100 K16  ; 触摸屏输入当前步骤
      MOV     D100 D98
      MRD
      AND     M425  ; 触摸屏左右臂切换
      AND<    D100 K20  ; 触摸屏输入当前步骤
      ADD     D100 K20 D98
      MPP
      RST     M380  ; 设置步骤序号
6925  LD      M194  ; 有其他在运行
      ZRST    M91 M92  ; 上一步 / 下一步
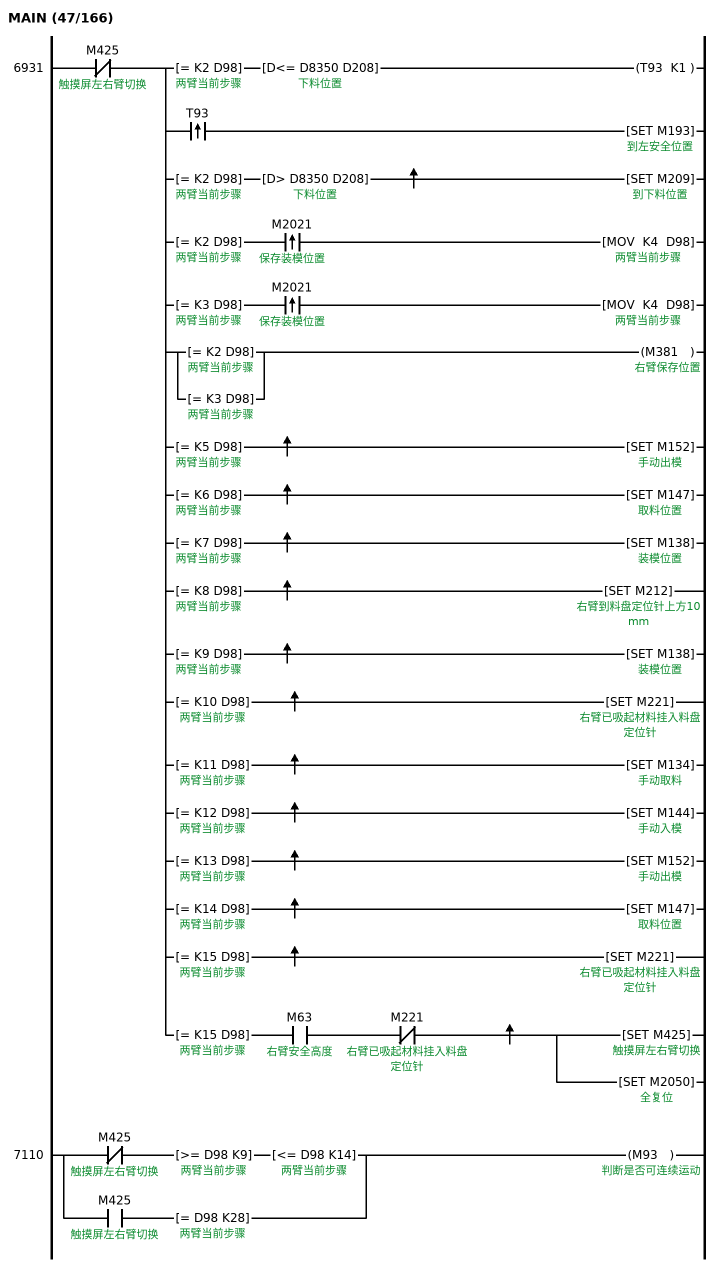
6931  LDI     M425  ; 触摸屏左右臂切换
      MPS
      AND=    K2 D98  ; 两臂当前步骤
      ANDD<=  D8350 D208  ; 下料位置
      OUT     T93 K1
      MRD
      ANDP    T93
      SET     M193  ; 到左安全位置
      MRD
      AND=    K2 D98  ; 两臂当前步骤
      ANDD>   D8350 D208  ; 下料位置
      MEP
      SET     M209  ; 到下料位置
      MRD
      AND=    K2 D98  ; 两臂当前步骤
      ANDP    M2021  ; 保存装模位置
      MOV     K4 D98
      MRD
      AND=    K3 D98  ; 两臂当前步骤
      ANDP    M2021  ; 保存装模位置
      MOV     K4 D98
      MRD
      LD=     K2 D98  ; 两臂当前步骤
      OR=     K3 D98  ; 两臂当前步骤
      ANB
      OUT     M381  ; 右臂保存位置
      MRD
      AND=    K5 D98  ; 两臂当前步骤
      MEP
      SET     M152  ; 手动出模
      MRD
      AND=    K6 D98  ; 两臂当前步骤
      MEP
      SET     M147  ; 取料位置
      MRD
      AND=    K7 D98  ; 两臂当前步骤
      MEP
      SET     M138  ; 装模位置
      MRD
      AND=    K8 D98  ; 两臂当前步骤
      MEP
      SET     M212  ; 右臂到料盘定位针上方10mm
      MRD
      AND=    K9 D98  ; 两臂当前步骤
      MEP
      SET     M138  ; 装模位置
      MRD
      AND=    K10 D98  ; 两臂当前步骤
      MEP
      SET     M221  ; 右臂已吸起材料挂入料盘定位针
      MRD
      AND=    K11 D98  ; 两臂当前步骤
      MEP
      SET     M134  ; 手动取料
      MRD
      AND=    K12 D98  ; 两臂当前步骤
      MEP
      SET     M144  ; 手动入模
      MRD
      AND=    K13 D98  ; 两臂当前步骤
      MEP
      SET     M152  ; 手动出模
      MRD
      AND=    K14 D98  ; 两臂当前步骤
      MEP
      SET     M147  ; 取料位置
      MRD
      AND=    K15 D98  ; 两臂当前步骤
      MEP
      SET     M221  ; 右臂已吸起材料挂入料盘定位针
      MPP
      AND=    K15 D98  ; 两臂当前步骤
      AND     M63  ; 右臂安全高度
      ANI     M221  ; 右臂已吸起材料挂入料盘定位针
      MEP
      SET     M425  ; 触摸屏左右臂切换
      SET     M2050  ; 全复位
7110  LDI     M425  ; 触摸屏左右臂切换
      AND>=   D98 K9  ; 两臂当前步骤
      AND<=   D98 K14  ; 两臂当前步骤
      LD      M425  ; 触摸屏左右臂切换
      AND=    D98 K28  ; 两臂当前步骤
      ORB
      OUT     M93  ; 判断是否可连续运动
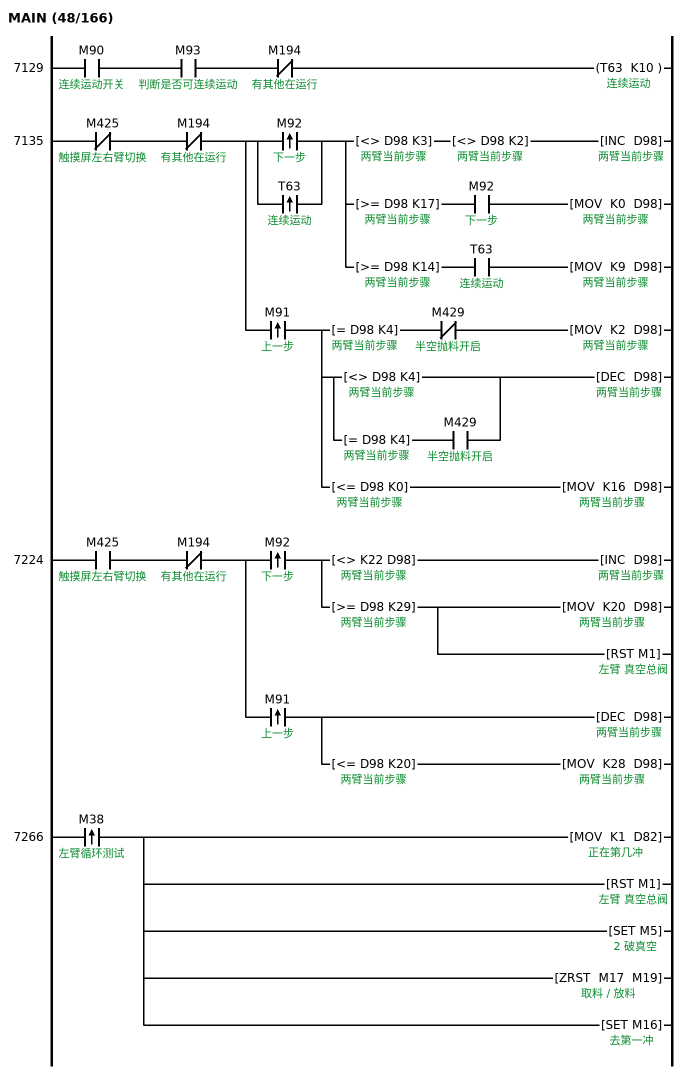
7129  LD      M90  ; 连续运动开关
      AND     M93  ; 判断是否可连续运动
      ANI     M194  ; 有其他在运行
      OUT     T63 K10  ; 连续运动
7135  LDI     M425  ; 触摸屏左右臂切换
      ANI     M194  ; 有其他在运行
      MPS
      LDP     M92  ; 下一步
      ORP     T63  ; 连续运动
      ANB
      MPS
      AND<>   D98 K3  ; 两臂当前步骤
      AND<>   D98 K2  ; 两臂当前步骤
      INC     D98
      MRD
      AND>=   D98 K17  ; 两臂当前步骤
      AND     M92  ; 下一步
      MOV     K0 D98
      MPP
      AND>=   D98 K14  ; 两臂当前步骤
      AND     T63  ; 连续运动
      MOV     K9 D98
      MPP
      ANDP    M91  ; 上一步
      MPS
      AND=    D98 K4  ; 两臂当前步骤
      ANI     M429  ; 半空抛料开启
      MOV     K2 D98
      MRD
      LD<>    D98 K4  ; 两臂当前步骤
      LD=     D98 K4  ; 两臂当前步骤
      AND     M429  ; 半空抛料开启
      ORB
      ANB
      DEC     D98
      MPP
      AND<=   D98 K0  ; 两臂当前步骤
      MOV     K16 D98
7224  LD      M425  ; 触摸屏左右臂切换
      ANI     M194  ; 有其他在运行
      MPS
      ANDP    M92  ; 下一步
      MPS
      AND<>   K22 D98  ; 两臂当前步骤
      INC     D98
      MPP
      AND>=   D98 K29  ; 两臂当前步骤
      MOV     K20 D98
      RST     M1  ; 左臂 真空总阀
      MPP
      ANDP    M91  ; 上一步
      DEC     D98
      AND<=   D98 K20  ; 两臂当前步骤
      MOV     K28 D98
7266  LDP     M38  ; 左臂循环测试
      MOV     K1 D82
      RST     M1  ; 左臂 真空总阀
      SET     M5  ; 2 破真空
      ZRST    M17 M19  ; 取料 / 放料
      SET     M16  ; 去第一冲
